(* PLC project SafeLOGIC-1, BrAutomation SafeDESIGNER  4.3.2.11 *)
(* stored: companyURL http://www.br-automation.com, creationDateTime Fri May 18 07:40:53 2018 *)

PROGRAM CheckAnalogSensor

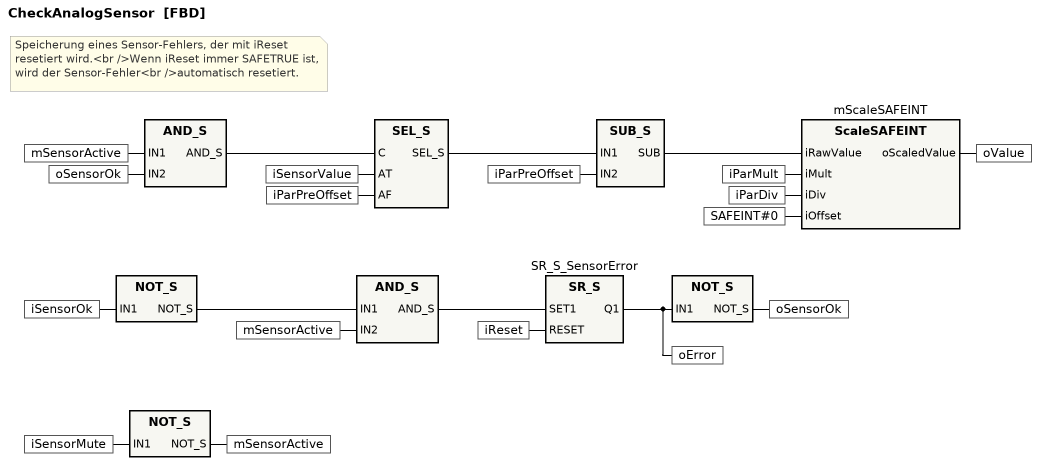
(* FBD diagram, written out as Structured Text *)
mSensorActive := NOT_S(iSensorMute);
(* Speicherung eines Sensor-Fehlers, der mit iReset resetiert wird.<br />Wenn iReset immer SAFETRUE ist, wird der Sensor-Fehler<br />automatisch resetiert. *)
SR_S_SensorError(SET1 := AND_S(NOT_S(iSensorOk), mSensorActive), RESET := iReset);
oSensorOk := NOT_S(SR_S_SensorError.Q1);
oError := SR_S_SensorError.Q1;
mScaleSAFEINT(iRawValue := SUB_S(SEL_S(AND_S(mSensorActive, oSensorOk), iSensorValue, iParPreOffset), iParPreOffset), iMult := iParMult, iDiv := iParDiv, iOffset := SAFEINT#0);
oValue := mScaleSAFEINT.oScaledValue;
END_PROGRAM
